{attribute 'GeneratedUsingTerminal: EL9183--0000'}
{attribute addProperty BoxType "EL9183--0000"}
{attribute addProperty Description "EL9183 Potential Connection, 1 x 16 contacts"}
{attribute addProperty Physics "KK"}
{attribute addProperty Id "EL9183"}
{attribute addProperty CRC "2253793365"}
{attribute addProperty Size "0"}
TYPE EL9183_86562855 EXTENDS EtcSlaveTerminalBase_947E5A46 :
STRUCT
END_STRUCT
END_TYPE

(* stored: Version 1.2.0.0, ProductVersion 3.1.4024.9
   DUT EL9183_86562855: Id {0c632c4c-8888-41f9-b233-adb62d6f3a4d} *)
